{attribute 'GeneratedUsingTerminal: EP9128-0020-0016'}
{attribute addProperty BoxType "EP9128-0020-0016"}
{attribute addProperty Description "EP9128-0020 8x EtherCAT junction"}
{attribute addProperty Physics "YYKY"}
{attribute addProperty Id "InfoDataAT %I*InfoData_6F19DB2B2"}
{attribute addProperty CRC "532711307"}
{attribute addProperty Size "2"}
TYPE EP9128_1FC0878B EXTENDS EtcSlaveBoxBase_77A0E4A7 :
STRUCT
	{attribute addProperty Name "InfoData"}
	InfoData : InfoData_6F19DB2B;
END_STRUCT
END_TYPE

(* stored: Version 1.2.0.0, ProductVersion 3.1.4024.11
   DUT EP9128_1FC0878B: Id {9b4dbc75-8af3-4ac2-80ea-27f53d9d4f59} *)
